FUNCTION_BLOCK FB_TimeDistance
VAR_INPUT
	bInitEvent			: BOOL;
	bEndEvent			: BOOL;
	tTimeout			: TIME := t#10s;
	tCurrentDistanceTime	: TIME;
	bResetCTU				: BOOL;
END_VAR
VAR_OUTPUT
	tRefDistanceTime				: TIME;
	bIntervalBelowRefTime			: BOOL;
	nIntervalBelowRefCounter		: INT;
	bIntervalAboveRefTime		: BOOL;
	nIntervalAboveRefCounter		: INT;
END_VAR
VAR

	tonRefDistance		: TON;
	rsRefDistance			: RS;
	aCTU				: ARRAY [1..2] OF CTU;

END_VAR

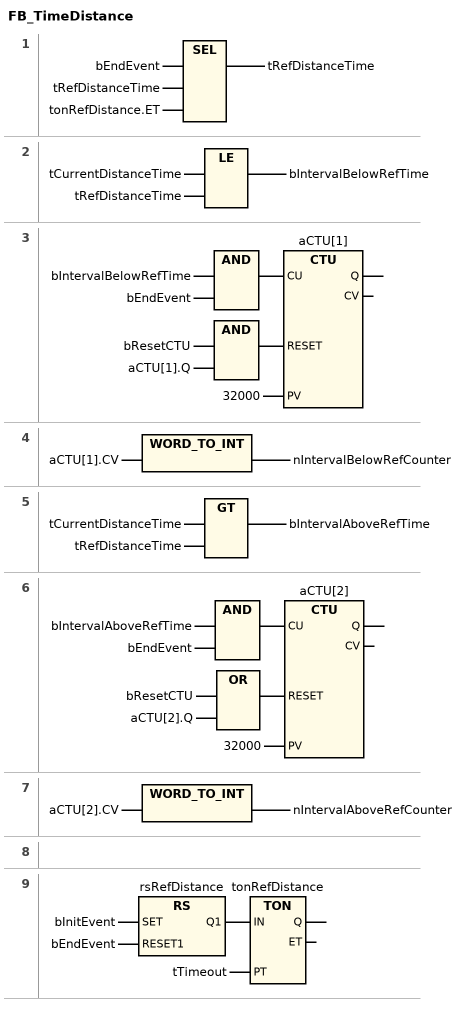
// NETWORK 1
tRefDistanceTime := SEL(bEndEvent, tRefDistanceTime, tonRefDistance.ET);

// NETWORK 2
bIntervalBelowRefTime := tCurrentDistanceTime <= tRefDistanceTime;

// NETWORK 3
aCTU[1](CU := bIntervalBelowRefTime AND bEndEvent, RESET := bResetCTU AND aCTU[1].Q, PV := 32000); // CTU

// NETWORK 4
nIntervalBelowRefCounter := WORD_TO_INT(aCTU[1].CV);

// NETWORK 5
bIntervalAboveRefTime := tCurrentDistanceTime > tRefDistanceTime;

// NETWORK 6
aCTU[2](CU := bIntervalAboveRefTime AND bEndEvent, RESET := bResetCTU OR aCTU[2].Q, PV := 32000); // CTU

// NETWORK 7
nIntervalAboveRefCounter := WORD_TO_INT(aCTU[2].CV);

// NETWORK 8

// NETWORK 9
rsRefDistance(SET := bInitEvent, RESET1 := bEndEvent); // RS
tonRefDistance(IN := rsRefDistance.Q1, PT := tTimeout); // TON

END_FUNCTION_BLOCK

(* stored: Version 1.1.0.1
   POU FB_TimeDistance: Id {72c2db9d-b68b-4efe-9da7-3886df98b9cc}, SpecialFunc None *)
